SUBAPPLICATION SServer (* Subapplication Type *)
  (* Standard: 61499-2 *)
  (* Version 1.0, 2019-07-02, dorofeev *)
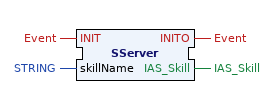
  EVENT_INPUT
    INIT; (* Initialization Request *)
  END_EVENT
  EVENT_OUTPUT
    INITO;
  END_EVENT
  VAR_INPUT
    skillName : STRING; (* Input event qualifier *)
  END_VAR
  PLUGS
    IAS_Skill : IAS_Skill;
  END_PLUGS
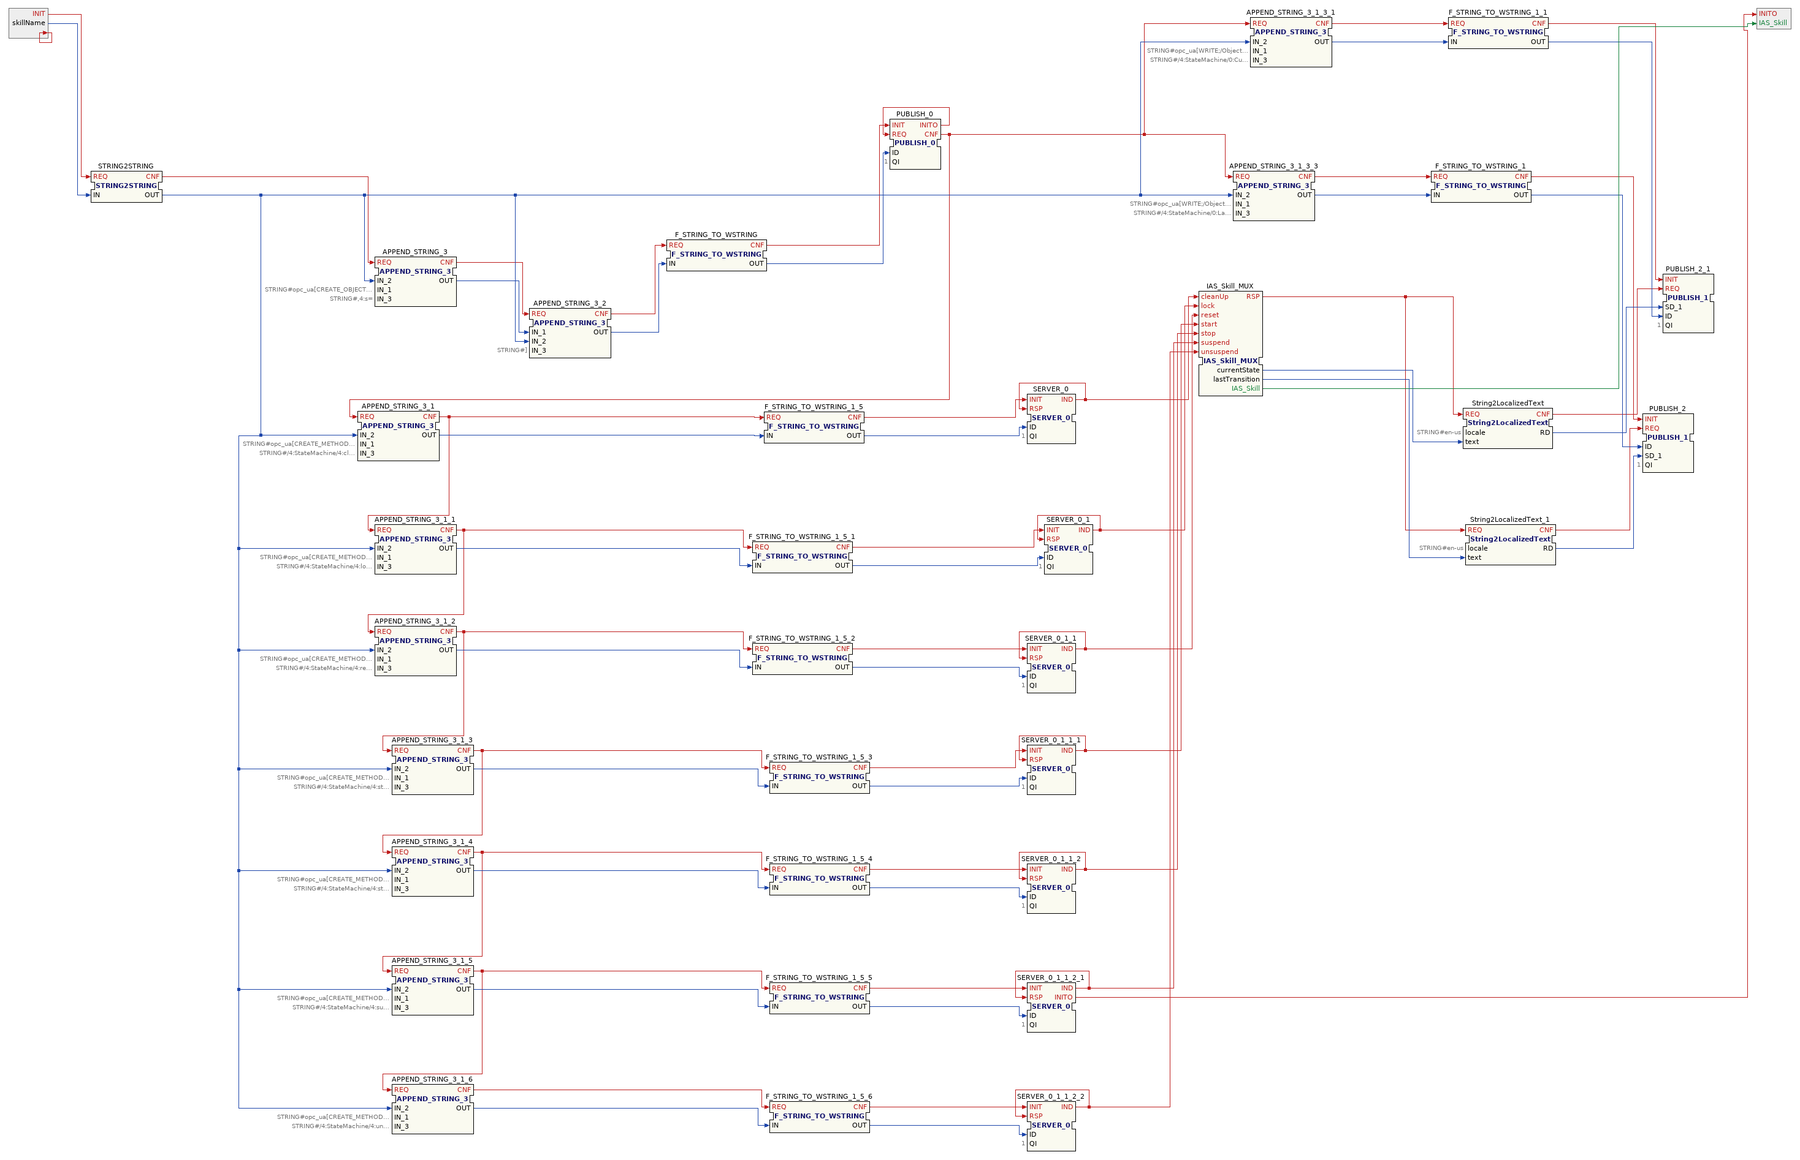
  FBS
    STRING2STRING : STRING2STRING;
    F_STRING_TO_WSTRING : F_STRING_TO_WSTRING;
    F_STRING_TO_WSTRING_1_5_2 : F_STRING_TO_WSTRING;
    APPEND_STRING_3_1_2 : APPEND_STRING_3(IN_1 := STRING#opc_ua[CREATE_METHOD;/Objects/4:skills/4:, IN_3 := STRING#/4:StateMachine/4:reset]);
    F_STRING_TO_WSTRING_1_5_3 : F_STRING_TO_WSTRING;
    F_STRING_TO_WSTRING_1_5_6 : F_STRING_TO_WSTRING;
    APPEND_STRING_3_1_1 : APPEND_STRING_3(IN_1 := STRING#opc_ua[CREATE_METHOD;/Objects/4:skills/4:, IN_3 := STRING#/4:StateMachine/4:lock]);
    APPEND_STRING_3 : APPEND_STRING_3(IN_1 := STRING#opc_ua[CREATE_OBJECT;,4:i=1002;/Objects/4:skills/4:, IN_3 := STRING#,4:s=);
    APPEND_STRING_3_1_6 : APPEND_STRING_3(IN_1 := STRING#opc_ua[CREATE_METHOD;/Objects/4:skills/4:, IN_3 := STRING#/4:StateMachine/4:unsuspend]);
    APPEND_STRING_3_1_5 : APPEND_STRING_3(IN_1 := STRING#opc_ua[CREATE_METHOD;/Objects/4:skills/4:, IN_3 := STRING#/4:StateMachine/4:suspend]);
    APPEND_STRING_3_1 : APPEND_STRING_3(IN_1 := STRING#opc_ua[CREATE_METHOD;/Objects/4:skills/4:, IN_3 := STRING#/4:StateMachine/4:cleanUp]);
    APPEND_STRING_3_1_4 : APPEND_STRING_3(IN_1 := STRING#opc_ua[CREATE_METHOD;/Objects/4:skills/4:, IN_3 := STRING#/4:StateMachine/4:stop]);
    F_STRING_TO_WSTRING_1_5_4 : F_STRING_TO_WSTRING;
    F_STRING_TO_WSTRING_1_5_1 : F_STRING_TO_WSTRING;
    F_STRING_TO_WSTRING_1_5_5 : F_STRING_TO_WSTRING;
    PUBLISH_0 : PUBLISH_0(QI := 1);
    F_STRING_TO_WSTRING_1_5 : F_STRING_TO_WSTRING;
    SERVER_0 : SERVER_0(QI := 1);
    SERVER_0_1 : SERVER_0(QI := 1);
    SERVER_0_1_1 : SERVER_0(QI := 1);
    SERVER_0_1_1_1 : SERVER_0(QI := 1);
    SERVER_0_1_1_2 : SERVER_0(QI := 1);
    SERVER_0_1_1_2_1 : SERVER_0(QI := 1);
    SERVER_0_1_1_2_2 : SERVER_0(QI := 1);
    String2LocalizedText : String2LocalizedText(locale := STRING#en-us);
    String2LocalizedText_1 : String2LocalizedText(locale := STRING#en-us);
    IAS_Skill_MUX : IAS_Skill_MUX;
    APPEND_STRING_3_1_3 : APPEND_STRING_3(IN_1 := STRING#opc_ua[CREATE_METHOD;/Objects/4:skills/4:, IN_3 := STRING#/4:StateMachine/4:start]);
    APPEND_STRING_3_1_3_1 : APPEND_STRING_3(IN_1 := STRING#opc_ua[WRITE;/Objects/4:skills/4:, IN_3 := STRING#/4:StateMachine/0:CurrentState]);
    APPEND_STRING_3_1_3_3 : APPEND_STRING_3(IN_1 := STRING#opc_ua[WRITE;/Objects/4:skills/4:, IN_3 := STRING#/4:StateMachine/0:LastTransition]);
    F_STRING_TO_WSTRING_1 : F_STRING_TO_WSTRING;
    PUBLISH_2 : PUBLISH_1(QI := 1);
    PUBLISH_2_1 : PUBLISH_1(QI := 1);
    F_STRING_TO_WSTRING_1_1 : F_STRING_TO_WSTRING;
    APPEND_STRING_3_2 : APPEND_STRING_3(IN_3 := STRING#]);
  END_FBS
  EVENT_CONNECTIONS
    INIT TO STRING2STRING.REQ;
    STRING2STRING.CNF TO APPEND_STRING_3.REQ;
    F_STRING_TO_WSTRING.CNF TO PUBLISH_0.INIT;
    PUBLISH_0.INITO TO PUBLISH_0.REQ;
    PUBLISH_0.CNF TO APPEND_STRING_3_1.REQ;
    APPEND_STRING_3_1.CNF TO APPEND_STRING_3_1_1.REQ;
    APPEND_STRING_3_1_1.CNF TO APPEND_STRING_3_1_2.REQ;
    APPEND_STRING_3_1_4.CNF TO APPEND_STRING_3_1_5.REQ;
    APPEND_STRING_3_1_5.CNF TO APPEND_STRING_3_1_6.REQ;
    F_STRING_TO_WSTRING_1_5.CNF TO SERVER_0.INIT;
    F_STRING_TO_WSTRING_1_5_1.CNF TO SERVER_0_1.INIT;
    F_STRING_TO_WSTRING_1_5_2.CNF TO SERVER_0_1_1.INIT;
    F_STRING_TO_WSTRING_1_5_3.CNF TO SERVER_0_1_1_1.INIT;
    F_STRING_TO_WSTRING_1_5_4.CNF TO SERVER_0_1_1_2.INIT;
    F_STRING_TO_WSTRING_1_5_5.CNF TO SERVER_0_1_1_2_1.INIT;
    F_STRING_TO_WSTRING_1_5_6.CNF TO SERVER_0_1_1_2_2.INIT;
     TO ;
     TO ;
     TO ;
     TO ;
     TO ;
     TO ;
     TO ;
    SERVER_0.IND TO SERVER_0.RSP;
    SERVER_0_1.IND TO SERVER_0_1.RSP;
    SERVER_0_1_1.IND TO SERVER_0_1_1.RSP;
    SERVER_0_1_1_1.IND TO SERVER_0_1_1_1.RSP;
    SERVER_0_1_1_2.IND TO SERVER_0_1_1_2.RSP;
    SERVER_0_1_1_2_1.IND TO SERVER_0_1_1_2_1.RSP;
    SERVER_0_1_1_2_2.IND TO SERVER_0_1_1_2_2.RSP;
    SERVER_0_1_1_2_1.INITO TO INITO;
    SERVER_0.IND TO IAS_Skill_MUX.cleanUp;
    SERVER_0_1.IND TO IAS_Skill_MUX.lock;
    SERVER_0_1_1.IND TO IAS_Skill_MUX.reset;
    SERVER_0_1_1_1.IND TO IAS_Skill_MUX.start;
    SERVER_0_1_1_2.IND TO IAS_Skill_MUX.stop;
    SERVER_0_1_1_2_1.IND TO IAS_Skill_MUX.suspend;
    SERVER_0_1_1_2_2.IND TO IAS_Skill_MUX.unsuspend;
    IAS_Skill_MUX.RSP TO String2LocalizedText.REQ;
    IAS_Skill_MUX.RSP TO String2LocalizedText_1.REQ;
    APPEND_STRING_3_1_3.CNF TO APPEND_STRING_3_1_4.REQ;
    APPEND_STRING_3_1_2.CNF TO APPEND_STRING_3_1_3.REQ;
    APPEND_STRING_3_1_3_3.CNF TO F_STRING_TO_WSTRING_1.REQ;
    F_STRING_TO_WSTRING_1.CNF TO PUBLISH_2.INIT;
    String2LocalizedText_1.CNF TO PUBLISH_2.REQ;
    APPEND_STRING_3_1_3_1.CNF TO F_STRING_TO_WSTRING_1_1.REQ;
    APPEND_STRING_3_1.CNF TO F_STRING_TO_WSTRING_1_5.REQ;
    APPEND_STRING_3_1_1.CNF TO F_STRING_TO_WSTRING_1_5_1.REQ;
    APPEND_STRING_3_1_2.CNF TO F_STRING_TO_WSTRING_1_5_2.REQ;
    APPEND_STRING_3_1_3.CNF TO F_STRING_TO_WSTRING_1_5_3.REQ;
    APPEND_STRING_3_1_4.CNF TO F_STRING_TO_WSTRING_1_5_4.REQ;
    APPEND_STRING_3_1_5.CNF TO F_STRING_TO_WSTRING_1_5_5.REQ;
    APPEND_STRING_3_1_6.CNF TO F_STRING_TO_WSTRING_1_5_6.REQ;
    APPEND_STRING_3.CNF TO APPEND_STRING_3_2.REQ;
    APPEND_STRING_3_2.CNF TO F_STRING_TO_WSTRING.REQ;
    PUBLISH_0.CNF TO APPEND_STRING_3_1_3_3.REQ;
    PUBLISH_0.CNF TO APPEND_STRING_3_1_3_1.REQ;
    F_STRING_TO_WSTRING_1_1.CNF TO PUBLISH_2_1.INIT;
    String2LocalizedText.CNF TO PUBLISH_2_1.REQ;
  END_CONNECTIONS
  DATA_CONNECTIONS
    skillName TO STRING2STRING.IN;
    STRING2STRING.OUT TO APPEND_STRING_3.IN_2;
    F_STRING_TO_WSTRING.OUT TO PUBLISH_0.ID;
    STRING2STRING.OUT TO APPEND_STRING_3_1.IN_2;
    STRING2STRING.OUT TO APPEND_STRING_3_1_1.IN_2;
    STRING2STRING.OUT TO APPEND_STRING_3_1_2.IN_2;
    STRING2STRING.OUT TO APPEND_STRING_3_1_4.IN_2;
    STRING2STRING.OUT TO APPEND_STRING_3_1_5.IN_2;
    STRING2STRING.OUT TO APPEND_STRING_3_1_6.IN_2;
    F_STRING_TO_WSTRING_1_5.OUT TO SERVER_0.ID;
    F_STRING_TO_WSTRING_1_5_1.OUT TO SERVER_0_1.ID;
    F_STRING_TO_WSTRING_1_5_2.OUT TO SERVER_0_1_1.ID;
    F_STRING_TO_WSTRING_1_5_3.OUT TO SERVER_0_1_1_1.ID;
    F_STRING_TO_WSTRING_1_5_4.OUT TO SERVER_0_1_1_2.ID;
    F_STRING_TO_WSTRING_1_5_5.OUT TO SERVER_0_1_1_2_1.ID;
    F_STRING_TO_WSTRING_1_5_6.OUT TO SERVER_0_1_1_2_2.ID;
    IAS_Skill_MUX.currentState TO String2LocalizedText.text;
    IAS_Skill_MUX.lastTransition TO String2LocalizedText_1.text;
    STRING2STRING.OUT TO APPEND_STRING_3_1_3.IN_2;
    STRING2STRING.OUT TO APPEND_STRING_3_1_3_1.IN_2;
    STRING2STRING.OUT TO APPEND_STRING_3_1_3_3.IN_2;
    APPEND_STRING_3_1_3_3.OUT TO F_STRING_TO_WSTRING_1.IN;
    F_STRING_TO_WSTRING_1.OUT TO PUBLISH_2.ID;
    String2LocalizedText_1.RD TO PUBLISH_2.SD_1;
    String2LocalizedText.RD TO PUBLISH_2_1.SD_1;
    APPEND_STRING_3_1_3_1.OUT TO F_STRING_TO_WSTRING_1_1.IN;
    F_STRING_TO_WSTRING_1_1.OUT TO PUBLISH_2_1.ID;
    APPEND_STRING_3_1.OUT TO F_STRING_TO_WSTRING_1_5.IN;
    APPEND_STRING_3_1_1.OUT TO F_STRING_TO_WSTRING_1_5_1.IN;
    APPEND_STRING_3_1_2.OUT TO F_STRING_TO_WSTRING_1_5_2.IN;
    APPEND_STRING_3_1_3.OUT TO F_STRING_TO_WSTRING_1_5_3.IN;
    APPEND_STRING_3_1_4.OUT TO F_STRING_TO_WSTRING_1_5_4.IN;
    APPEND_STRING_3_1_5.OUT TO F_STRING_TO_WSTRING_1_5_5.IN;
    APPEND_STRING_3_1_6.OUT TO F_STRING_TO_WSTRING_1_5_6.IN;
    APPEND_STRING_3.OUT TO APPEND_STRING_3_2.IN_1;
    STRING2STRING.OUT TO APPEND_STRING_3_2.IN_2;
    APPEND_STRING_3_2.OUT TO F_STRING_TO_WSTRING.IN;
  END_CONNECTIONS
  ADAPTER_CONNECTIONS
    IAS_Skill_MUX.IAS_Skill TO IAS_Skill;
  END_CONNECTIONS
END_SUBAPPLICATION
